{attribute 'GeneratedUsingTerminal: EP1816-0008-0018'}
{attribute addProperty BoxType "EP1816-0008-0018"}
{attribute addProperty Id "InputAT %I*ARRAY[0..7] OF BOOL8Sync_ErrorAT %I*BOOL1"}
{attribute addProperty CRC "2788215981"}
{attribute addProperty Size "9"}
TYPE DIG_Inputs_Channel_CC455148 :
STRUCT
	{attribute addProperty Name "Input"}
	Input AT %I* : ARRAY[0..7] OF BOOL;
	{attribute addProperty Name "Sync_Error"}
	Sync_Error AT %I* : BOOL;
END_STRUCT
END_TYPE

(* stored: Version 1.2.0.0, ProductVersion 3.1.4024.9
   DUT DIG_Inputs_Channel_CC455148: Id {5e2fdce4-974b-42af-8590-a9e676a2e01a} *)
